(* CoDeSys 2.3 export: FTURNONK15PUMP.EXP *)

(* POU K15/fTurnOnK15Pump, ST *)
FUNCTION fTurnOnK15Pump :BOOL
VAR_INPUT
	PumpID : USINT;
END_VAR
VAR
END_VAR
fSetK15Pump(TRUE, PumpID);
END_FUNCTION
